{attribute addProperty BoxType "EK1100-0000-0018"}
{attribute addProperty Id "Beckhoff_EK11xxEK1122Beckhoff_EK11xxEK1122_0F9A188531439.25A_0018_EK1110_0043_0016EK1110_179A0949162A_0024_EK1122_0008_0016EK1122_179A0949162A_0023_EK1122_0000_0018EK1122_179A0949162A_0022_EK1122_0000_0017EK1122_179A0949162A_0021_EK1122_0000_0016EK1122_179A0949162A_0020_EK1121_0010_0016EK1121_179A0949162A_0019_EK1110_0044_0016EK1110_179A0949162A_0017_EK1110_0008_0016EK1110_179A0949162A_0016_EK1110_0000_0017EK1110_179A0949162A_0015_EK1110_0000_0016EK1110_179A0949162A_0014_EK1110_0000_0000EK1110_179A0949162"}
{attribute addProperty CRC "3240383487"}
{attribute addProperty SizeInBites "490"}
{attribute addProperty SizeInBytes "61.25"}
TYPE Beckhoff_EK11xx_C12453FF EXTENDS EK1100_179A0949 :
STRUCT
	{attribute addProperty Name "Beckhoff_EK11xxEK1122"}
	Beckhoff_EK11xxEK1122 : Beckhoff_EK11xxEK1122_0F9A1885;
	{attribute addProperty Name "A_0018_EK1110_0043_0016"}
	A_0018_EK1110_0043_0016 : EK1110_179A0949;
	{attribute addProperty Name "A_0024_EK1122_0008_0016"}
	A_0024_EK1122_0008_0016 : EK1122_179A0949;
	{attribute addProperty Name "A_0023_EK1122_0000_0018"}
	A_0023_EK1122_0000_0018 : EK1122_179A0949;
	{attribute addProperty Name "A_0022_EK1122_0000_0017"}
	A_0022_EK1122_0000_0017 : EK1122_179A0949;
	{attribute addProperty Name "A_0021_EK1122_0000_0016"}
	A_0021_EK1122_0000_0016 : EK1122_179A0949;
	{attribute addProperty Name "A_0020_EK1121_0010_0016"}
	A_0020_EK1121_0010_0016 : EK1121_179A0949;
	{attribute addProperty Name "A_0019_EK1110_0044_0016"}
	A_0019_EK1110_0044_0016 : EK1110_179A0949;
	{attribute addProperty Name "A_0017_EK1110_0008_0016"}
	A_0017_EK1110_0008_0016 : EK1110_179A0949;
	{attribute addProperty Name "A_0016_EK1110_0000_0017"}
	A_0016_EK1110_0000_0017 : EK1110_179A0949;
	{attribute addProperty Name "A_0015_EK1110_0000_0016"}
	A_0015_EK1110_0000_0016 : EK1110_179A0949;
	{attribute addProperty Name "A_0014_EK1110_0000_0000"}
	A_0014_EK1110_0000_0000 : EK1110_179A0949;
END_STRUCT
END_TYPE

(* stored: Version 1.2.0.0, ProductVersion 3.1.4024.9
   DUT Beckhoff_EK11xx_C12453FF: Id {bb84ff64-6075-4394-9312-6daea364cee4} *)
